FUNCTION_BLOCK fb_dsopenclose
VAR_INPUT
END_VAR
VAR_OUTPUT
END_VAR
VAR
	ax1: AXIS_REF;
	McJog: MC_Jog;
	McPower: MC_Power;
	McReset: MC_Reset;
	McStop: MC_Stop;
	iState: INT;
END_VAR

(*McPower(Axis := ax1, Enable := TRUE, Enable_Positive := TRUE, Enable_Negative := TRUE);
McReset(Axis := ax1);
McJog(Axis := ax1);
CASE iState OF 
	0: 
		iState := 10;
	
	10:
		McReset(Axis:= ax1, Execute := TRUE);
		IF McReset.Done THEN
			iState := 20;
		ELSIF McReset.Error THEN
			iState := 999;
		END_IF
	
	20:
		IF McPower.Status THEN
			iState := 30;
		END_IF
		
	30:
		IF engage.stepopen OR DSin.open THEN
			cntrlstate.cover_moving := TRUE;
			McJog(Axis := ax1, JogForward := NOT DSin.endStopBck, Velocity := 20);
			IF DSin.endStopBck THEN
				cntrlstate.cover_moving := FALSE;
				engage.stepper := FALSE;
				engage.stepopen := FALSE;
				DSin.open := FALSE;
			END_IF
		ELSIF engage.stepclose OR DSin.close THEN
			cntrlstate.cover_moving := TRUE;
			McJog(Axis := ax1, JogBackwards := NOT DSin.endStopFrnt, Velocity := 20);
			IF DSin.endStopFrnt THEN
				cntrlstate.cover_moving := FALSE;
				engage.stepper := FALSE;
				engage.stepclose := FALSE;
				DSin.close := FALSE;
			END_IF
		END_IF
END_CASE
*)
IF engage.stepopen OR DSin.open THEN
	cntrlstate.cover_moving := TRUE;
	DSout.servoBackward := TRUE;
	IF DSin.endStopBck = FALSE THEN
		DSout.servoBackward := FALSE;
		cntrlstate.cover_moving := FALSE;
		engage.stepper := FALSE;
		engage.stepopen := FALSE;
		DSin.open := FALSE;
	END_IF
ELSIF engage.stepclose OR DSin.close THEN
	cntrlstate.cover_moving := TRUE;
	DSout.servoForward := TRUE;
	IF DSin.endStopFrnt = FALSE THEN
		DSout.servoForward := FALSE;
		cntrlstate.cover_moving := FALSE;
		engage.stepper := FALSE;
		engage.stepclose := FALSE;
		DSin.close := FALSE;
	END_IF
END_IF

END_FUNCTION_BLOCK

(* stored: Version 1.1.0.1, ProductVersion 3.1.4024.5
   POU fb_dsopenclose: Id {84a8c466-db40-4d05-ad00-947b96fbc127}, SpecialFunc None *)
